TYPE ST_CAMERA_Performance :
STRUCT
	tLastDiff 		: TIME;
	tAverageDiff 	: TIME;
	arrTimeDiff 	: ARRAY[0..9] OF TIME;
END_STRUCT
END_TYPE

(* stored: Version 1.1.0.1
   DUT ST_CAMERA_Performance: Id {5b782c9f-2d0d-4067-a680-0aea995a5d7d} *)
